Fanuc KAREL source: kt00518.KL

-- PROVISIONAL review KL for V770-1; original PC SHA256 c716fd2537f54d96e523011930b79b47a94d258f79cccf6786ad681fd4968269
-- Incomplete behavior may be omitted. Consult companion uncertainty JSON. Do not deploy.
PROGRAM KT00518
%NOLOCKGROUP
VAR
  OUT : BOOLEAN
-- UNRESOLVED_DECL P1 type=000106
-- UNRESOLVED_DECL P2 type=000102
BEGIN
  -- UNRESOLVED_PC offsets 5-20; opcodes 2E,22,32,35
  -- UNRESOLVED_PC offsets 25-40; opcodes 2E,22,32,35
  -- UNRESOLVED_PC offsets 45-78; opcodes 49,7E,49,7E,AC,23
  -- UNRESOLVED_PC offsets 83-87; opcodes 7F
END KT00518
